// ============================================================================
// GlobalVars.db - 边框缓存机全局变量数据块
// ============================================================================
// 功能说明:
//   定义 DJ-2026-005 边框缓存机 PLC 控制系统的所有全局变量.
//   作为 OB1 主程序与各功能块之间的数据交换中心, 实现统一的数据管理.
//
// 数据组织:
//   - stGlobal:        全局控制信号和系统状态 (来自FB_2001_CommonAlarm)
//   - stExternal:      外部设备交互信号 (组框机/打胶机/机器人)
//   - stConveyor:      四层输送机系统信号 (含4层数组, ARRAY[1..4])
//   - stPickPlace:     取放料机构信号 (含4卡槽调度与接料安全互锁)
//   - stRecipeManager: 10组配方存储池与当前生效配方
//   - stFeeder:        打胶机送料机构信号 (X2台车4卡槽物料检测)
//   - astServoAxis:    3轴伺服控制数组 (Z/X1/X2)
// ============================================================================

DATA_BLOCK GlobalVars

VAR
    // =========================================================================
    // 第一部分: 全局控制信号与系统状态 (FB_2001_CommonAlarm)
    // =========================================================================
    stGlobal   : ST_CommonAlarm;

    // =========================================================================
    // 第二部分: 外部设备交互信号 (ST_ExternalDevice)
    // =========================================================================
    stExternal : ST_ExternalDevice;

    // =========================================================================
    // 第三部分: 四层输送机系统信号 (ST_SingleLayerConveyor ARRAY[1..4])
    // =========================================================================
    stConveyor : STRUCT
        astLayer                 : ARRAY[1..4] OF ST_SingleLayerConveyor;
        i_bAutoMode              : BOOL := FALSE;    // 自动运行模式
        i_bManualMode            : BOOL := FALSE;    // 手动调试模式
        i_bStart                 : BOOL := FALSE;    // 自动循环启动
        i_bStop                  : BOOL := FALSE;    // 停止
        i_dSeparateTimeoutMs     : DINT := 5000;     // 分料超时时间(ms)
        i_dDebounceMs            : DINT := 0;        // 传感器消抖(ms)
        i_bSafetyDoorOk          : BOOL := TRUE;     // 安全门OK
        i_bVfdFault              : BOOL := FALSE;    // 变频器故障
        q_bRunning               : BOOL := FALSE;    // 4层 OR
        q_bFault                 : BOOL := FALSE;    // 4层 OR
        q_iAlarmCode             : INT := 0;         // 4层报警码 MIN
    END_STRUCT;

    // =========================================================================
    // 第四部分: 取放料机构信号与10组配方管理器
    // =========================================================================
    stPickPlace      : ST_PickPlace;
    stRecipeManager  : ST_RecipeManager;

    // =========================================================================
    // 第五部分: 打胶机送料机构信号 (ST_GlueFeeder)
    // =========================================================================
    stFeeder         : ST_GlueFeeder;

    // =========================================================================
    // 第五部分B: 伺服轴数组 (ST_ServoAxis V3.0, PLCopen MC Part 1)
    // 轴索引: [1]=Z轴(升降) [2]=X1轴(取放料横移) [3]=X2轴(打胶机送料)
    // =========================================================================
    astServoAxis     : ARRAY[1..3] OF ST_ServoAxis;

    // =========================================================================
    // 第六部分: 功能块实例
    // =========================================================================
    fbExternalDevice      : FB_ExternalDeviceInteraction;
    fbConveyor_L1         : FB_1002_SingleLayerConveyor_BufferFraming;
    fbConveyor_L2         : FB_1002_SingleLayerConveyor_BufferFraming;
    fbConveyor_L3         : FB_1002_SingleLayerConveyor_BufferFraming;
    fbConveyor_L4         : FB_1002_SingleLayerConveyor_BufferFraming;
    fbPickPlace           : FB_1003_PickPlace_BufferFraming;
    fbGlueFeeder          : FB_1004_GlueMachineFeeder_BufferFraming;
    fbCommonAlarm         : FB_2001_CommonAlarm_AllStation;
END_VAR

END_DATA_BLOCK
